{attribute addProperty BoxType "EL2535-0000-0021"}
{attribute addProperty Id "PWM_Status_ChannelAT %I*ARRAY[0..1] OF PWM_Status_Channel_789699B53240PWM_Control_ChannelAT %Q*ARRAY[0..1] OF PWM_Control_Channel_253BEA616480WcStateAT %I*WcState_F855686C1620InfoDataAT %I*InfoData_BC63D37F80100"}
{attribute addProperty CRC "4195700234"}
{attribute addProperty SizeInBites "192"}
{attribute addProperty SizeInBytes "24"}
TYPE EL2535_9AC04402 :
STRUCT
	{attribute addProperty Name "PWM_Status_Channel"}
	PWM_Status_Channel : ARRAY[0..1] OF PWM_Status_Channel_789699B5;
	{attribute addProperty Name "PWM_Control_Channel"}
	PWM_Control_Channel : ARRAY[0..1] OF PWM_Control_Channel_253BEA61;
	{attribute addProperty Name "WcState"}
	WcState : WcState_F855686C;
	{attribute addProperty Name "InfoData"}
	InfoData : InfoData_BC63D37F;
END_STRUCT
END_TYPE

(* stored: Version 1.2.0.0, ProductVersion 3.1.4024.9
   DUT EL2535_9AC04402: Id {bfbe0c4e-fb9f-42ed-9ead-fc2531349141} *)
